FUNCTION_BLOCK base 
VAR_INPUT
END_VAR
VAR_OUTPUT
END_VAR
VAR
	field1 : INT := 555;
END_VAR

METHOD METH : STRING
VAR_INPUT
END_VAR
METH := 'base';
END_METHOD

END_FUNCTION_BLOCK

(* stored: Version 1.1.0.1, ProductVersion 3.1.4022.10
   POU base: Id {4bdf7bb1-2c95-4efa-aeb8-c2bd9c7d66fd}, SpecialFunc None
   Method METH: Id {3ea16346-5c9b-4274-a1db-2e36b12f445a} *)
